//{{V2}}
ORGANIZATION_BLOCK OB1
TITLE= "Zyklisches Hauptprogramm"


AUTHOR:nb
FAMILY:nb
NAME:nb
VERSION:1.0


VAR_TEMP
       OB1_EV_CLASS:BYTE //Bits 0-3 = 1 (Coming event), Bits 4-7 = 1 (Event class 1)
       OB1_SCAN_1:BYTE //1 (Cold restart scan 1 of OB 1), 3 (Scan 2-n of OB 1)
       OB1_PRIORITY:BYTE //1 (Priority of 1 is lowest)
       OB1_OB_NUMBR:BYTE //1 (Organization block 1, OB1)
       OB1_RESERVED_1:BYTE //Reserved for system
       OB1_RESERVED_2:BYTE //Reserved for system
       OB1_PREV_CYCLE:INT //Cycle time of previous OB1 scan (milliseconds)
       OB1_MIN_CYCLE:INT //Minimum cycle time of OB1 (milliseconds)
       OB1_MAX_CYCLE:INT //Maximum cycle time of OB1 (milliseconds)
       OB1_DATE_TIME:DATE_AND_TIME //Date and time OB1 started
END_VAR
BEGIN

NETWORK
TITLE=
//{{a}}


       UN   M         0.0
       SPBN set
       S    M         0.0

       L    0
       T    LW        0
_for:  NOP  0

       L    LW        0
       L    P#        2.0
       *D
       T    LD       10


       AUF  DB       10
       L    LW        0
       ITD
       DTR
       EXP
       RND
       L    10
       MOD

       T    DBW [LD10]



       L    LW        0
       L    1
       +D
       T    LW        0


       L    LW        0
       L    10
       <I
       SPB  _for
NETWORK
TITLE=
//{{a}}


set:   NOP  0

       CALL FC       10
         links:=0
         rechts:=1
END_ORGANIZATION_BLOCK
